FUNCTION_BLOCK deserializeByteArray2LrealArray (* Basic Function Block Type *)
  (* Standard: 61499-2 *)
  (* Version 0.0, 19/09/2015, kollger, nxtControl GmbH, Template *)
  PACKAGE Main;
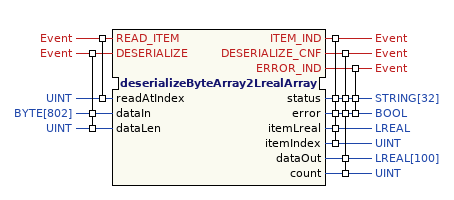
  EVENT_INPUT
    READ_ITEM WITH readAtIndex;
    DESERIALIZE WITH dataIn, dataLen; (* Normal Execution Request *)
  END_EVENT
  EVENT_OUTPUT
    ITEM_IND WITH itemLreal, itemIndex, status, error;
    DESERIALIZE_CNF WITH dataOut, count, status, error; (* Execution Confirmation *)
    ERROR_IND WITH status, error;
  END_EVENT
  VAR_INPUT
    readAtIndex : UINT;
    dataIn : ARRAY [0..801] OF BYTE;
    dataLen : UINT;
  END_VAR
  VAR_OUTPUT
    status : STRING[32];
    error : BOOL;
    itemLreal : LREAL;
    itemIndex : UINT;
    dataOut : ARRAY [0..99] OF LREAL;
    count : UINT;
  END_VAR
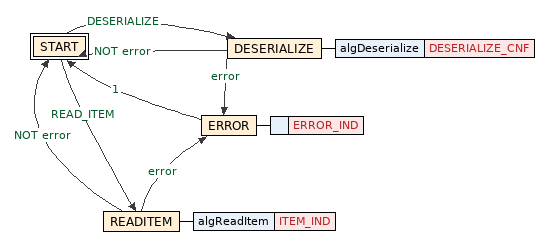
  EC_STATES
    START; (* Initial State *)
    DESERIALIZE : algDeserialize -> DESERIALIZE_CNF; (* Normal execution *)
    READITEM : algReadItem -> ITEM_IND;
    ERROR : -> ERROR_IND;
  END_STATES
  EC_TRANSITIONS
    START TO DESERIALIZE := DESERIALIZE;
    DESERIALIZE TO START := NOT error;
    START TO READITEM := READ_ITEM;
    READITEM TO START := NOT error;
    DESERIALIZE TO ERROR := error;
    ERROR TO START := 1;
    READITEM TO ERROR := error;
  END_TRANSITIONS
  ALGORITHM algDeserialize IN ST: (* Normally executed algorithm *)
VAR
	index : UINT := 0;
	byteindex : UINT := 0;
  mergeLWORD : LWORD := 16#0;
END_VAR;

IF dataLen <= 802 THEN

	(* read count length *)
	mergeLWORD := 16#0;
	mergeLWORD := mergeLWORD OR dataIn[0];
	mergeLWORD := SHL(mergeLWORD, 8);
	mergeLWORD := mergeLWORD OR dataIn[1];
	count := LWORD_TO_UINT(mergeLWORD);

  IF dataLen < (count * 8 + 2) THEN

  	(* Iterate through the BYTE array and transfer it to the LREAL ARRAY *)
  	FOR index := 0 TO count - 1 DO
  		mergeLWORD := 16#0;
  		byteindex := index * 8 + 2;
  		mergeLWORD := mergeLWORD OR dataIn[byteindex];
  		mergeLWORD := SHL(mergeLWORD, 8);
  		mergeLWORD := mergeLWORD OR dataIn[byteindex + 1];
  		mergeLWORD := SHL(mergeLWORD, 8);
  		mergeLWORD := mergeLWORD OR dataIn[byteindex + 2];
  		mergeLWORD := SHL(mergeLWORD, 8);
  		mergeLWORD := mergeLWORD OR dataIn[byteindex + 3];
  		mergeLWORD := SHL(mergeLWORD, 8);
  		mergeLWORD := mergeLWORD OR dataIn[byteindex + 4];
  		mergeLWORD := SHL(mergeLWORD, 8);
  		mergeLWORD := mergeLWORD OR dataIn[byteindex + 5];
  		mergeLWORD := SHL(mergeLWORD, 8);
  		mergeLWORD := mergeLWORD OR dataIn[byteindex + 6];
  		mergeLWORD := SHL(mergeLWORD, 8);
  		mergeLWORD := mergeLWORD OR dataIn[byteindex + 7];
  		dataOut[index] := DWORD_TO_LREAL(mergeLWORD);
  	END_FOR;
  	FOR index := index TO 99 DO
  		dataOut[index] := 0.0;
  	END_FOR;

  	error := FALSE;
  	status := STRING#'Ok';

  ELSE

    error := TRUE;
  	status := STRING#'dataIn invalid size';

  END_IF;

ELSE
  error := TRUE;
  status := STRING#'dataIn to big';
END_IF;
  END_ALGORITHM
  ALGORITHM algReadItem IN ST:
IF readAtIndex <= count THEN

  itemLreal := dataOut[readAtIndex];
  itemIndex := readAtIndex;

  error := FALSE;
  status := STRING#'Ok';
ELSE
  itemLreal := 0.0;
  itemIndex := 0;
  error := TRUE;
  status := STRING#'Read out of range';
END_IF;
;
  END_ALGORITHM
END_FUNCTION_BLOCK
